SUBAPPLICATION Uebung_225_AXA (* Dreieck-Sollwertmarker (wie 225, aber ein reiner Adapter-Spiegel: NumericValue_PHYSA, AR_ADD_2, AR_TO_AI, Q_ChildPosition_AI, Q_NumericValue_PHYSA) *)
  (* Standard: 61499-2; Description: Copyright (c) 2026 Meisterschulen am Ostbahnhof This program and the accompanying materials are made available under the terms of the Eclipse Public License 2.0 which is available at https://www.eclipse.org/legal/epl-2.0/ SPDX-License-Identifier: EPL-2.0 *)
  (* Version 1.1, 2026-09-06, Franz Höpfinger, Meisterschulen am Ostbahnhof, Enable xScale on Q_ChildPosition_Dreieck *)
  (* Version 1.0, 2026-09-05, Franz Höpfinger, Meisterschulen am Ostbahnhof, pure-adapter mirror of Uebung_225_AX: NumericValue_PHYSA/AR_SPLIT_2/AR_ADD_2/initval_AR/AR_TO_AI/initval_AI/Q_ChildPosition_AI/Q_NumericValue_PHYSA - no plain Event/DataConnections at all *)
  PACKAGE Uebungen;
  IMPORT Uebungen::const::UT::Dreieck::DefaultPool_Dreieck::Polygon_Bargraph_Mittelmarker;
  IMPORT Uebungen::const::UT::Dreieck::DefaultPool_Dreieck::Container_Sollwertmarker;
  IMPORT Uebungen::const::UT::Dreieck::DefaultPool_Dreieck_Numeric::NumberVariable_Sollwert_N;
  IMPORT Uebungen::const::UT::Dreieck::DefaultPool_Dreieck_Numeric::NumberVariable_Istwert_N;
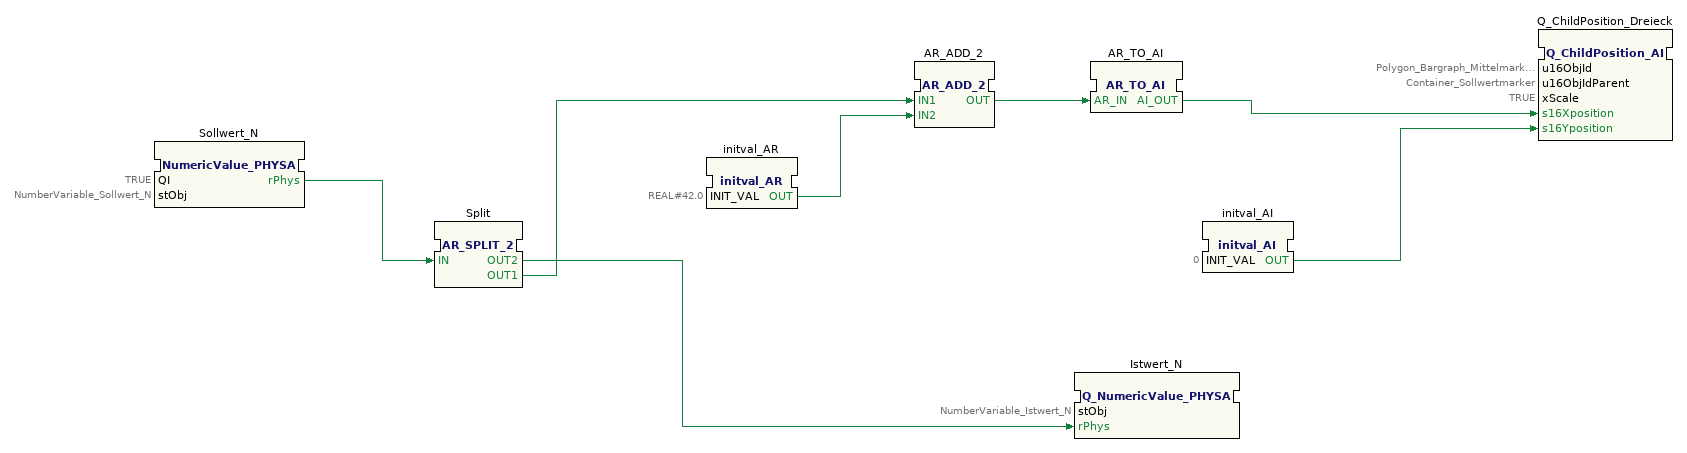
  FBS
    Sollwert_N : isobus::UT::io::NumericValue::NumericValue_PHYSA(QI := TRUE, stObj := NumberVariable_Sollwert_N);
    Split : adapter::events::unidirectional::AR_SPLIT_2;
    Istwert_N : isobus::UT::Q::Q_NumericValue_PHYSA(stObj := NumberVariable_Istwert_N);
    AR_ADD_2 : adapter::iec61131::arithmetic::AR_ADD_2;
    initval_AR : adapter::types::unidirectional::AR::initval::initval_AR(INIT_VAL := REAL#42.0);
    AR_TO_AI : adapter::conversion::unidirectional::AR_TO_AI;
    Q_ChildPosition_Dreieck : isobus::UT::Q::Q_ChildPosition_AI(u16ObjId := Polygon_Bargraph_Mittelmarker, u16ObjIdParent := Container_Sollwertmarker, xScale := TRUE);
    initval_AI : adapter::types::unidirectional::AI::initval::initval_AI(INIT_VAL := 0);
  END_FBS
  ADAPTER_CONNECTIONS
    Sollwert_N.rPhys TO Split.IN;
    Split.OUT2 TO Istwert_N.rPhys;
    Split.OUT1 TO AR_ADD_2.IN1;
    initval_AR.OUT TO AR_ADD_2.IN2;
    AR_ADD_2.OUT TO AR_TO_AI.AR_IN;
    AR_TO_AI.AI_OUT TO Q_ChildPosition_Dreieck.s16Xposition;
    initval_AI.OUT TO Q_ChildPosition_Dreieck.s16Yposition;
  END_CONNECTIONS
END_SUBAPPLICATION
